// TIA Portal V15.1 export
// export: Created 2024-05-17T05:38:59.8000198Z, ExportSetting WithDefaults, DisplayName Totally Integrated Automation Portal, DisplayVersion V15.1 Update 5, DisplayName TIA Portal Openness, DisplayVersion V15.1 Update 5, DisplayName SINAMICS Startdrive Advanced, DisplayVersion V15.1, DisplayName G130, G150, S120, S150, SINAMICS MV, S210, DisplayVersion V15.1, DisplayName G110M, G120, G120C, G120D, G120P, DisplayVersion V15.1, DisplayName STEP 7 Professional, DisplayVersion V15.1 Update 5, DisplayName STEP 7 Safety, DisplayVersion V15.1, DisplayName WinCC Professional, DisplayVersion V15.1 Update 5, DisplayName SIMATIC Visualization Architect, DisplayVersion V15.1
FUNCTION "209000NCP01Config" : Void   // FC290, FBD
TITLE = 209000NCP01Config
{ S7_Optimized_Access := 'FALSE' }
AUTHOR : VCC
VERSION : 0.1
// stored: AutoNumber false, IsIECCheckEnabled false, SetENOAutomatically False, UDAEnableTagReadback false
BEGIN

REGION Network 1: **** --------------------- ETA Fuses --------------------- ****
END_REGION

REGION Network 2: **** 4.2 - Machine Status - Parameters **** AE01-JC31 // Fuse Module 1..8 (Fuse 1-16)
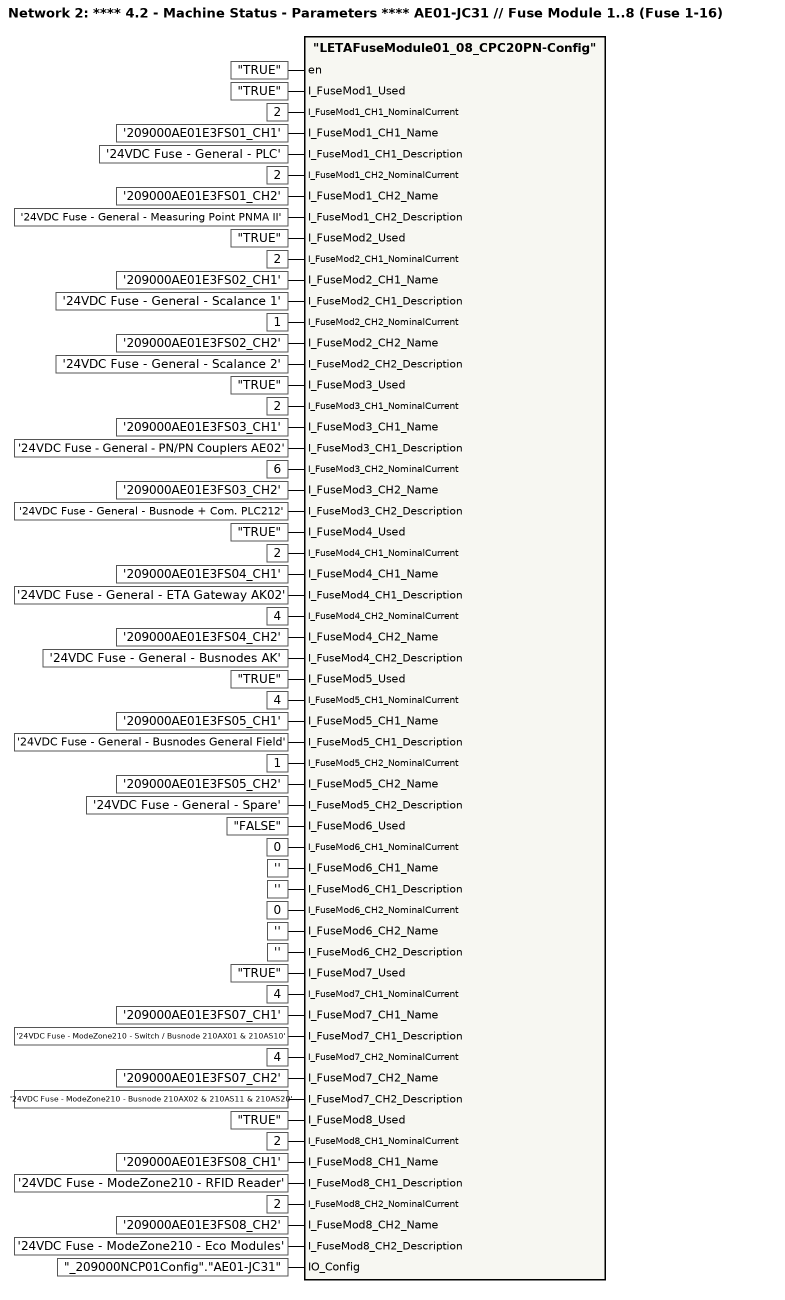
   IF "TRUE" THEN
       "LETAFuseModule01_08_CPC20PN-Config"(I_FuseMod1_Used := "TRUE",
                               I_FuseMod1_CH1_NominalCurrent := 2,
                               I_FuseMod1_CH1_Name := '209000AE01E3FS01_CH1',
                               I_FuseMod1_CH1_Description := '24VDC Fuse - General - PLC',
                               I_FuseMod1_CH2_NominalCurrent := 2,
                               I_FuseMod1_CH2_Name := '209000AE01E3FS01_CH2',
                               I_FuseMod1_CH2_Description := '24VDC Fuse - General - Measuring Point PNMA II',
                               I_FuseMod2_Used := "TRUE",
                               I_FuseMod2_CH1_NominalCurrent := 2,
                               I_FuseMod2_CH1_Name := '209000AE01E3FS02_CH1',
                               I_FuseMod2_CH1_Description := '24VDC Fuse - General - Scalance 1',
                               I_FuseMod2_CH2_NominalCurrent := 1,
                               I_FuseMod2_CH2_Name := '209000AE01E3FS02_CH2',
                               I_FuseMod2_CH2_Description := '24VDC Fuse - General - Scalance 2',
                               I_FuseMod3_Used := "TRUE",
                               I_FuseMod3_CH1_NominalCurrent := 2,
                               I_FuseMod3_CH1_Name := '209000AE01E3FS03_CH1',
                               I_FuseMod3_CH1_Description := '24VDC Fuse - General - PN/PN Couplers AE02',
                               I_FuseMod3_CH2_NominalCurrent := 6,
                               I_FuseMod3_CH2_Name := '209000AE01E3FS03_CH2',
                               I_FuseMod3_CH2_Description := '24VDC Fuse - General - Busnode + Com. PLC212',
                               I_FuseMod4_Used := "TRUE",
                               I_FuseMod4_CH1_NominalCurrent := 2,
                               I_FuseMod4_CH1_Name := '209000AE01E3FS04_CH1',
                               I_FuseMod4_CH1_Description := '24VDC Fuse - General - ETA Gateway AK02',
                               I_FuseMod4_CH2_NominalCurrent := 4,
                               I_FuseMod4_CH2_Name := '209000AE01E3FS04_CH2',
                               I_FuseMod4_CH2_Description := '24VDC Fuse - General - Busnodes AK',
                               I_FuseMod5_Used := "TRUE",
                               I_FuseMod5_CH1_NominalCurrent := 4,
                               I_FuseMod5_CH1_Name := '209000AE01E3FS05_CH1',
                               I_FuseMod5_CH1_Description := '24VDC Fuse - General - Busnodes General Field',
                               I_FuseMod5_CH2_NominalCurrent := 1,
                               I_FuseMod5_CH2_Name := '209000AE01E3FS05_CH2',
                               I_FuseMod5_CH2_Description := '24VDC Fuse - General - Spare',
                               I_FuseMod6_Used := "FALSE",
                               I_FuseMod6_CH1_NominalCurrent := 0,
                               I_FuseMod6_CH1_Name := '',
                               I_FuseMod6_CH1_Description := '',
                               I_FuseMod6_CH2_NominalCurrent := 0,
                               I_FuseMod6_CH2_Name := '',
                               I_FuseMod6_CH2_Description := '',
                               I_FuseMod7_Used := "TRUE",
                               I_FuseMod7_CH1_NominalCurrent := 4,
                               I_FuseMod7_CH1_Name := '209000AE01E3FS07_CH1',
                               I_FuseMod7_CH1_Description := '24VDC Fuse - ModeZone210 - Switch / Busnode 210AX01 & 210AS10',
                               I_FuseMod7_CH2_NominalCurrent := 4,
                               I_FuseMod7_CH2_Name := '209000AE01E3FS07_CH2',
                               I_FuseMod7_CH2_Description := '24VDC Fuse - ModeZone210 - Busnode 210AX02 & 210AS11 & 210AS20',
                               I_FuseMod8_Used := "TRUE",
                               I_FuseMod8_CH1_NominalCurrent := 2,
                               I_FuseMod8_CH1_Name := '209000AE01E3FS08_CH1',
                               I_FuseMod8_CH1_Description := '24VDC Fuse - ModeZone210 - RFID Reader',
                               I_FuseMod8_CH2_NominalCurrent := 2,
                               I_FuseMod8_CH2_Name := '209000AE01E3FS08_CH2',
                               I_FuseMod8_CH2_Description := '24VDC Fuse - ModeZone210 - Eco Modules',
                               IO_Config := "_209000NCP01Config"."AE01-JC31");
   END_IF;
END_REGION

REGION Network 3: **** 4.2 - Machine Status - Parameters **** AE01-JC31 // Fuse Module 9..16 (Fuse 17-32)
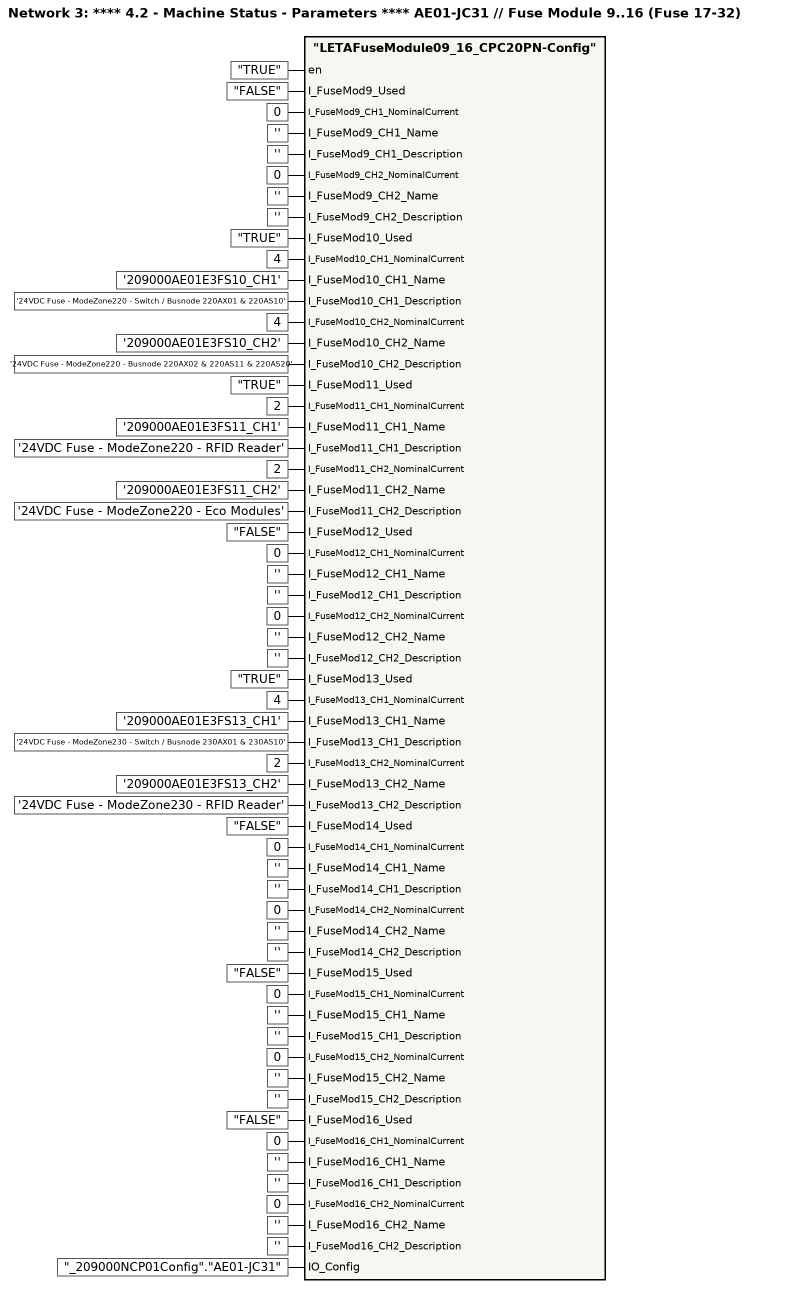
   IF "TRUE" THEN
       "LETAFuseModule09_16_CPC20PN-Config"(I_FuseMod9_Used := "FALSE",
                               I_FuseMod9_CH1_NominalCurrent := 0,
                               I_FuseMod9_CH1_Name := '',
                               I_FuseMod9_CH1_Description := '',
                               I_FuseMod9_CH2_NominalCurrent := 0,
                               I_FuseMod9_CH2_Name := '',
                               I_FuseMod9_CH2_Description := '',
                               I_FuseMod10_Used := "TRUE",
                               I_FuseMod10_CH1_NominalCurrent := 4,
                               I_FuseMod10_CH1_Name := '209000AE01E3FS10_CH1',
                               I_FuseMod10_CH1_Description := '24VDC Fuse - ModeZone220 - Switch / Busnode 220AX01 & 220AS10',
                               I_FuseMod10_CH2_NominalCurrent := 4,
                               I_FuseMod10_CH2_Name := '209000AE01E3FS10_CH2',
                               I_FuseMod10_CH2_Description := '24VDC Fuse - ModeZone220 - Busnode 220AX02 & 220AS11 & 220AS20',
                               I_FuseMod11_Used := "TRUE",
                               I_FuseMod11_CH1_NominalCurrent := 2,
                               I_FuseMod11_CH1_Name := '209000AE01E3FS11_CH1',
                               I_FuseMod11_CH1_Description := '24VDC Fuse - ModeZone220 - RFID Reader',
                               I_FuseMod11_CH2_NominalCurrent := 2,
                               I_FuseMod11_CH2_Name := '209000AE01E3FS11_CH2',
                               I_FuseMod11_CH2_Description := '24VDC Fuse - ModeZone220 - Eco Modules',
                               I_FuseMod12_Used := "FALSE",
                               I_FuseMod12_CH1_NominalCurrent := 0,
                               I_FuseMod12_CH1_Name := '',
                               I_FuseMod12_CH1_Description := '',
                               I_FuseMod12_CH2_NominalCurrent := 0,
                               I_FuseMod12_CH2_Name := '',
                               I_FuseMod12_CH2_Description := '',
                               I_FuseMod13_Used := "TRUE",
                               I_FuseMod13_CH1_NominalCurrent := 4,
                               I_FuseMod13_CH1_Name := '209000AE01E3FS13_CH1',
                               I_FuseMod13_CH1_Description := '24VDC Fuse - ModeZone230 - Switch / Busnode 230AX01 & 230AS10',
                               I_FuseMod13_CH2_NominalCurrent := 2,
                               I_FuseMod13_CH2_Name := '209000AE01E3FS13_CH2',
                               I_FuseMod13_CH2_Description := '24VDC Fuse - ModeZone230 - RFID Reader',
                               I_FuseMod14_Used := "FALSE",
                               I_FuseMod14_CH1_NominalCurrent := 0,
                               I_FuseMod14_CH1_Name := '',
                               I_FuseMod14_CH1_Description := '',
                               I_FuseMod14_CH2_NominalCurrent := 0,
                               I_FuseMod14_CH2_Name := '',
                               I_FuseMod14_CH2_Description := '',
                               I_FuseMod15_Used := "FALSE",
                               I_FuseMod15_CH1_NominalCurrent := 0,
                               I_FuseMod15_CH1_Name := '',
                               I_FuseMod15_CH1_Description := '',
                               I_FuseMod15_CH2_NominalCurrent := 0,
                               I_FuseMod15_CH2_Name := '',
                               I_FuseMod15_CH2_Description := '',
                               I_FuseMod16_Used := "FALSE",
                               I_FuseMod16_CH1_NominalCurrent := 0,
                               I_FuseMod16_CH1_Name := '',
                               I_FuseMod16_CH1_Description := '',
                               I_FuseMod16_CH2_NominalCurrent := 0,
                               I_FuseMod16_CH2_Name := '',
                               I_FuseMod16_CH2_Description := '',
                               IO_Config := "_209000NCP01Config"."AE01-JC31");
   END_IF;
END_REGION

REGION Network 4: **** 4.2 - Machine Status - Parameters **** AK02-JC32 // Fuse Module 1..8 (Fuse 1-16)
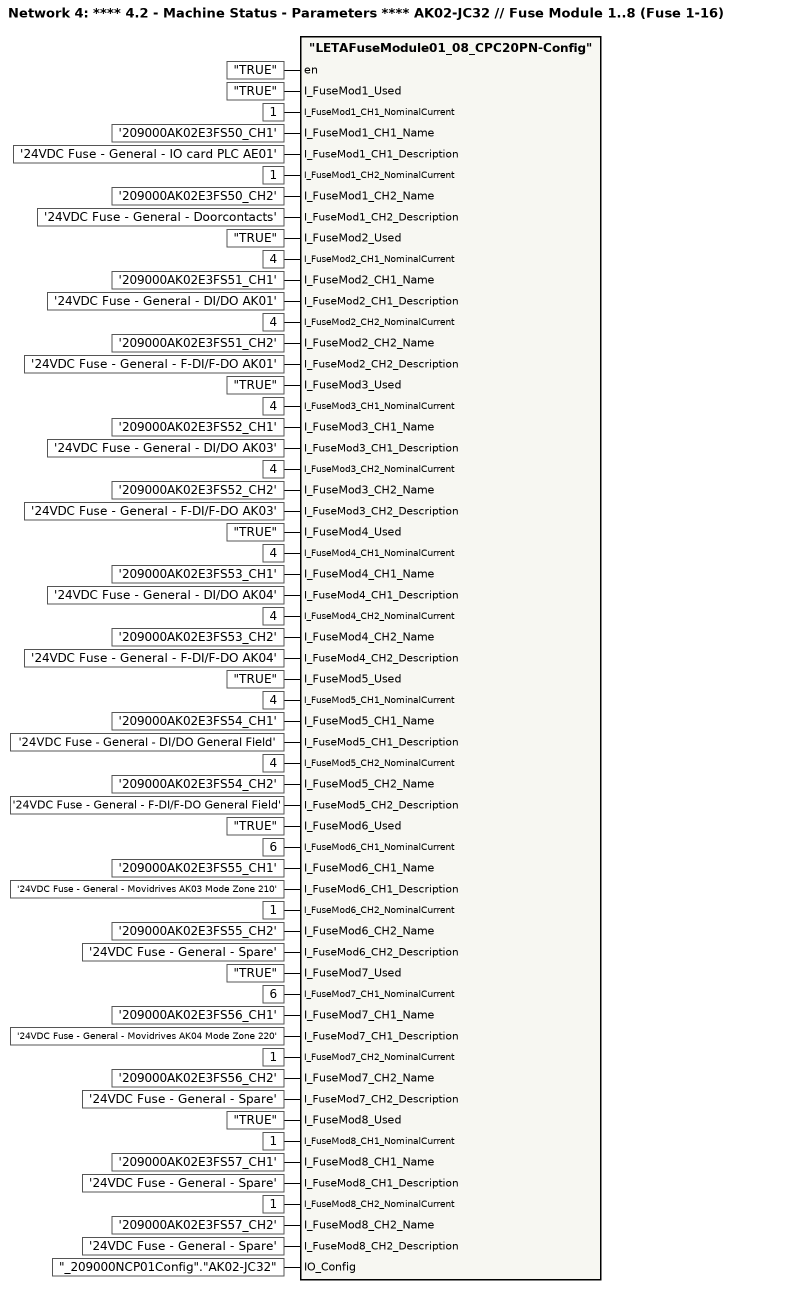
   IF "TRUE" THEN
       "LETAFuseModule01_08_CPC20PN-Config"(I_FuseMod1_Used := "TRUE",
                               I_FuseMod1_CH1_NominalCurrent := 1,
                               I_FuseMod1_CH1_Name := '209000AK02E3FS50_CH1',
                               I_FuseMod1_CH1_Description := '24VDC Fuse - General - IO card PLC AE01',
                               I_FuseMod1_CH2_NominalCurrent := 1,
                               I_FuseMod1_CH2_Name := '209000AK02E3FS50_CH2',
                               I_FuseMod1_CH2_Description := '24VDC Fuse - General - Doorcontacts',
                               I_FuseMod2_Used := "TRUE",
                               I_FuseMod2_CH1_NominalCurrent := 4,
                               I_FuseMod2_CH1_Name := '209000AK02E3FS51_CH1',
                               I_FuseMod2_CH1_Description := '24VDC Fuse - General - DI/DO AK01',
                               I_FuseMod2_CH2_NominalCurrent := 4,
                               I_FuseMod2_CH2_Name := '209000AK02E3FS51_CH2',
                               I_FuseMod2_CH2_Description := '24VDC Fuse - General - F-DI/F-DO AK01',
                               I_FuseMod3_Used := "TRUE",
                               I_FuseMod3_CH1_NominalCurrent := 4,
                               I_FuseMod3_CH1_Name := '209000AK02E3FS52_CH1',
                               I_FuseMod3_CH1_Description := '24VDC Fuse - General - DI/DO AK03',
                               I_FuseMod3_CH2_NominalCurrent := 4,
                               I_FuseMod3_CH2_Name := '209000AK02E3FS52_CH2',
                               I_FuseMod3_CH2_Description := '24VDC Fuse - General - F-DI/F-DO AK03',
                               I_FuseMod4_Used := "TRUE",
                               I_FuseMod4_CH1_NominalCurrent := 4,
                               I_FuseMod4_CH1_Name := '209000AK02E3FS53_CH1',
                               I_FuseMod4_CH1_Description := '24VDC Fuse - General - DI/DO AK04',
                               I_FuseMod4_CH2_NominalCurrent := 4,
                               I_FuseMod4_CH2_Name := '209000AK02E3FS53_CH2',
                               I_FuseMod4_CH2_Description := '24VDC Fuse - General - F-DI/F-DO AK04',
                               I_FuseMod5_Used := "TRUE",
                               I_FuseMod5_CH1_NominalCurrent := 4,
                               I_FuseMod5_CH1_Name := '209000AK02E3FS54_CH1',
                               I_FuseMod5_CH1_Description := '24VDC Fuse - General - DI/DO General Field',
                               I_FuseMod5_CH2_NominalCurrent := 4,
                               I_FuseMod5_CH2_Name := '209000AK02E3FS54_CH2',
                               I_FuseMod5_CH2_Description := '24VDC Fuse - General - F-DI/F-DO General Field',
                               I_FuseMod6_Used := "TRUE",
                               I_FuseMod6_CH1_NominalCurrent := 6,
                               I_FuseMod6_CH1_Name := '209000AK02E3FS55_CH1',
                               I_FuseMod6_CH1_Description := '24VDC Fuse - General - Movidrives AK03 Mode Zone 210',
                               I_FuseMod6_CH2_NominalCurrent := 1,
                               I_FuseMod6_CH2_Name := '209000AK02E3FS55_CH2',
                               I_FuseMod6_CH2_Description := '24VDC Fuse - General - Spare',
                               I_FuseMod7_Used := "TRUE",
                               I_FuseMod7_CH1_NominalCurrent := 6,
                               I_FuseMod7_CH1_Name := '209000AK02E3FS56_CH1',
                               I_FuseMod7_CH1_Description := '24VDC Fuse - General - Movidrives AK04 Mode Zone 220',
                               I_FuseMod7_CH2_NominalCurrent := 1,
                               I_FuseMod7_CH2_Name := '209000AK02E3FS56_CH2',
                               I_FuseMod7_CH2_Description := '24VDC Fuse - General - Spare',
                               I_FuseMod8_Used := "TRUE",
                               I_FuseMod8_CH1_NominalCurrent := 1,
                               I_FuseMod8_CH1_Name := '209000AK02E3FS57_CH1',
                               I_FuseMod8_CH1_Description := '24VDC Fuse - General - Spare',
                               I_FuseMod8_CH2_NominalCurrent := 1,
                               I_FuseMod8_CH2_Name := '209000AK02E3FS57_CH2',
                               I_FuseMod8_CH2_Description := '24VDC Fuse - General - Spare',
                               IO_Config := "_209000NCP01Config"."AK02-JC32");
   END_IF;
END_REGION

REGION Network 5: **** 4.2 - Machine Status - Parameters **** AK02-JC32 // Fuse Module 9..16 (Fuse 17-32)
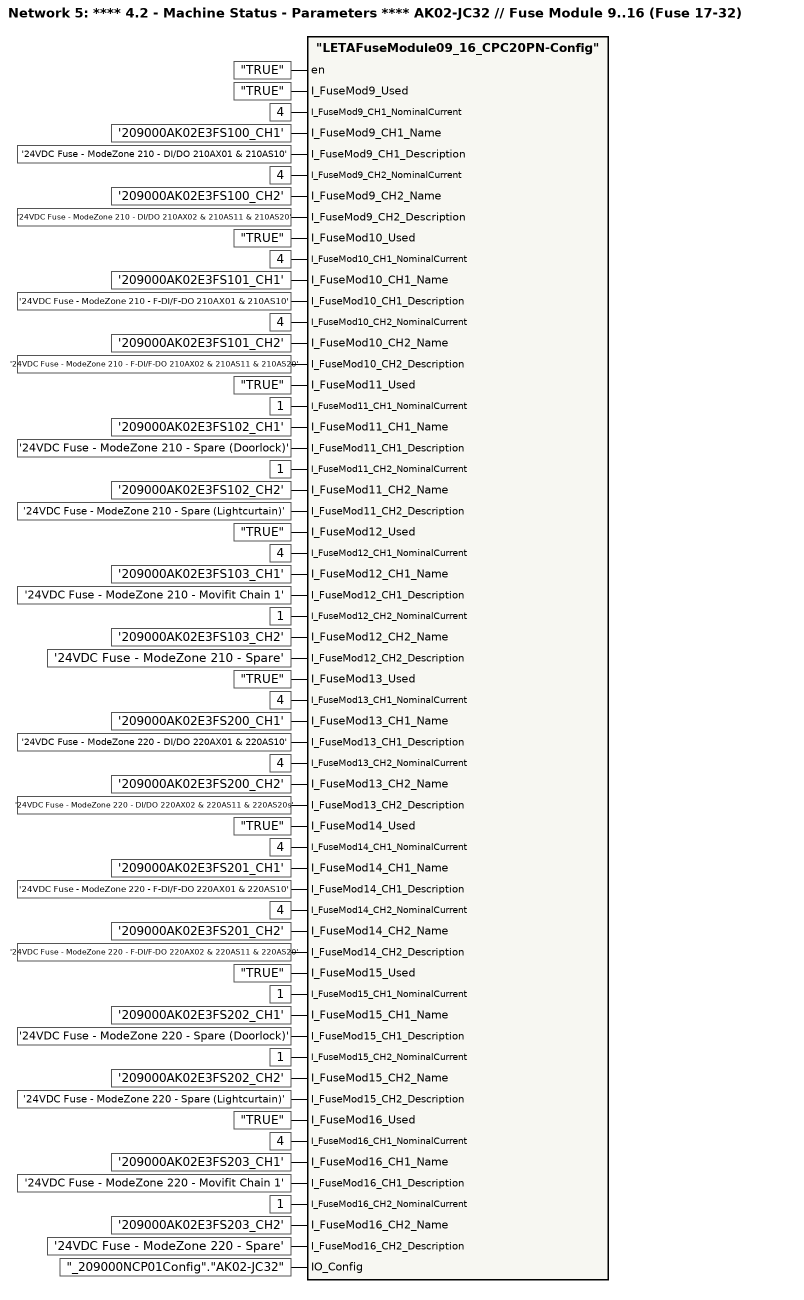
   IF "TRUE" THEN
       "LETAFuseModule09_16_CPC20PN-Config"(I_FuseMod9_Used := "TRUE",
                               I_FuseMod9_CH1_NominalCurrent := 4,
                               I_FuseMod9_CH1_Name := '209000AK02E3FS100_CH1',
                               I_FuseMod9_CH1_Description := '24VDC Fuse - ModeZone 210 - DI/DO 210AX01 & 210AS10',
                               I_FuseMod9_CH2_NominalCurrent := 4,
                               I_FuseMod9_CH2_Name := '209000AK02E3FS100_CH2',
                               I_FuseMod9_CH2_Description := '24VDC Fuse - ModeZone 210 - DI/DO 210AX02 & 210AS11 & 210AS20',
                               I_FuseMod10_Used := "TRUE",
                               I_FuseMod10_CH1_NominalCurrent := 4,
                               I_FuseMod10_CH1_Name := '209000AK02E3FS101_CH1',
                               I_FuseMod10_CH1_Description := '24VDC Fuse - ModeZone 210 - F-DI/F-DO 210AX01 & 210AS10',
                               I_FuseMod10_CH2_NominalCurrent := 4,
                               I_FuseMod10_CH2_Name := '209000AK02E3FS101_CH2',
                               I_FuseMod10_CH2_Description := '24VDC Fuse - ModeZone 210 - F-DI/F-DO 210AX02 & 210AS11 & 210AS20',
                               I_FuseMod11_Used := "TRUE",
                               I_FuseMod11_CH1_NominalCurrent := 1,
                               I_FuseMod11_CH1_Name := '209000AK02E3FS102_CH1',
                               I_FuseMod11_CH1_Description := '24VDC Fuse - ModeZone 210 - Spare (Doorlock)',
                               I_FuseMod11_CH2_NominalCurrent := 1,
                               I_FuseMod11_CH2_Name := '209000AK02E3FS102_CH2',
                               I_FuseMod11_CH2_Description := '24VDC Fuse - ModeZone 210 - Spare (Lightcurtain)',
                               I_FuseMod12_Used := "TRUE",
                               I_FuseMod12_CH1_NominalCurrent := 4,
                               I_FuseMod12_CH1_Name := '209000AK02E3FS103_CH1',
                               I_FuseMod12_CH1_Description := '24VDC Fuse - ModeZone 210 - Movifit Chain 1',
                               I_FuseMod12_CH2_NominalCurrent := 1,
                               I_FuseMod12_CH2_Name := '209000AK02E3FS103_CH2',
                               I_FuseMod12_CH2_Description := '24VDC Fuse - ModeZone 210 - Spare',
                               I_FuseMod13_Used := "TRUE",
                               I_FuseMod13_CH1_NominalCurrent := 4,
                               I_FuseMod13_CH1_Name := '209000AK02E3FS200_CH1',
                               I_FuseMod13_CH1_Description := '24VDC Fuse - ModeZone 220 - DI/DO 220AX01 & 220AS10',
                               I_FuseMod13_CH2_NominalCurrent := 4,
                               I_FuseMod13_CH2_Name := '209000AK02E3FS200_CH2',
                               I_FuseMod13_CH2_Description := '24VDC Fuse - ModeZone 220 - DI/DO 220AX02 & 220AS11 & 220AS20s',
                               I_FuseMod14_Used := "TRUE",
                               I_FuseMod14_CH1_NominalCurrent := 4,
                               I_FuseMod14_CH1_Name := '209000AK02E3FS201_CH1',
                               I_FuseMod14_CH1_Description := '24VDC Fuse - ModeZone 220 - F-DI/F-DO 220AX01 & 220AS10',
                               I_FuseMod14_CH2_NominalCurrent := 4,
                               I_FuseMod14_CH2_Name := '209000AK02E3FS201_CH2',
                               I_FuseMod14_CH2_Description := '24VDC Fuse - ModeZone 220 - F-DI/F-DO 220AX02 & 220AS11 & 220AS20',
                               I_FuseMod15_Used := "TRUE",
                               I_FuseMod15_CH1_NominalCurrent := 1,
                               I_FuseMod15_CH1_Name := '209000AK02E3FS202_CH1',
                               I_FuseMod15_CH1_Description := '24VDC Fuse - ModeZone 220 - Spare (Doorlock)',
                               I_FuseMod15_CH2_NominalCurrent := 1,
                               I_FuseMod15_CH2_Name := '209000AK02E3FS202_CH2',
                               I_FuseMod15_CH2_Description := '24VDC Fuse - ModeZone 220 - Spare (Lightcurtain)',
                               I_FuseMod16_Used := "TRUE",
                               I_FuseMod16_CH1_NominalCurrent := 4,
                               I_FuseMod16_CH1_Name := '209000AK02E3FS203_CH1',
                               I_FuseMod16_CH1_Description := '24VDC Fuse - ModeZone 220 - Movifit Chain 1',
                               I_FuseMod16_CH2_NominalCurrent := 1,
                               I_FuseMod16_CH2_Name := '209000AK02E3FS203_CH2',
                               I_FuseMod16_CH2_Description := '24VDC Fuse - ModeZone 220 - Spare',
                               IO_Config := "_209000NCP01Config"."AK02-JC32");
   END_IF;
END_REGION

REGION Network 6: **** 4.2 - Machine Status - Parameters **** AK02-JC32 // Fuse Module 17..24 (Fuse 33-48)
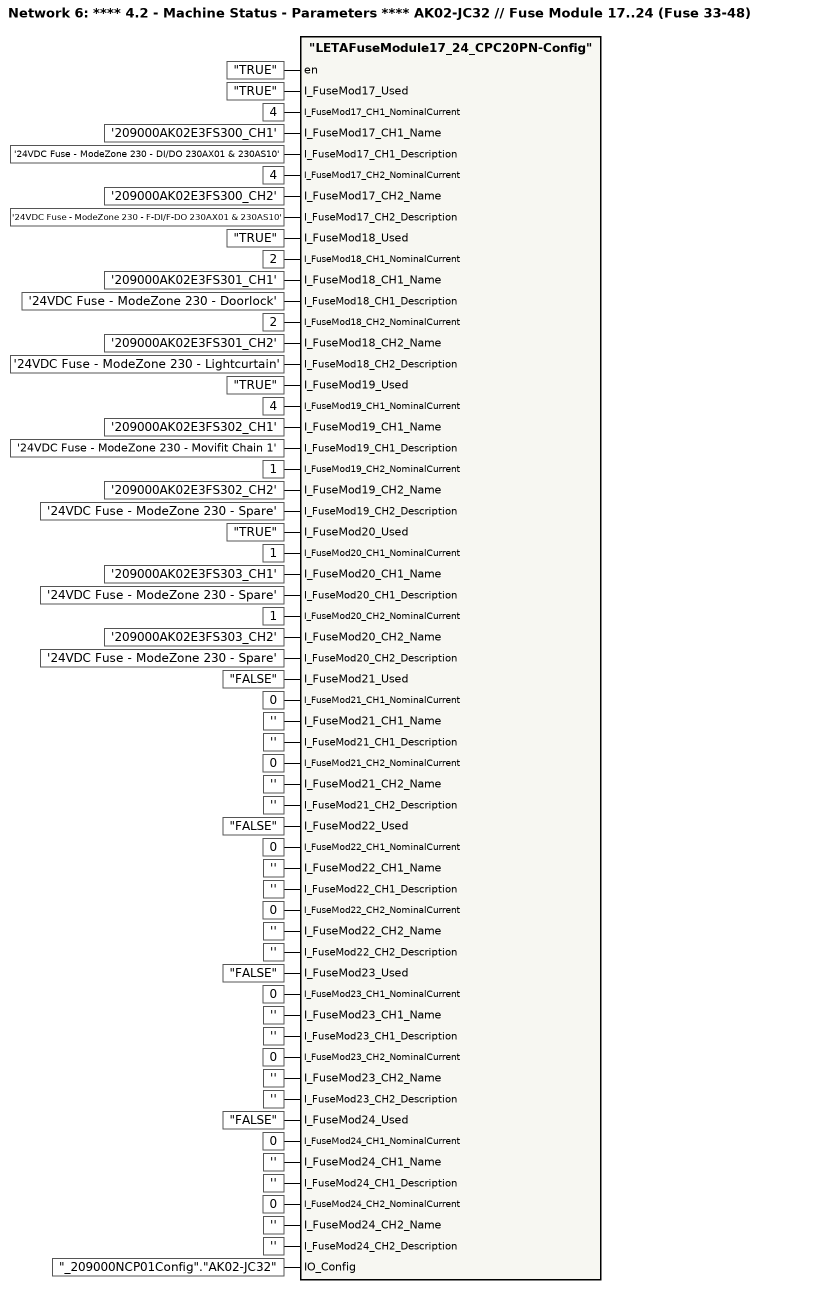
   IF "TRUE" THEN
       "LETAFuseModule17_24_CPC20PN-Config"(I_FuseMod17_Used := "TRUE",
                               I_FuseMod17_CH1_NominalCurrent := 4,
                               I_FuseMod17_CH1_Name := '209000AK02E3FS300_CH1',
                               I_FuseMod17_CH1_Description := '24VDC Fuse - ModeZone 230 - DI/DO 230AX01 & 230AS10',
                               I_FuseMod17_CH2_NominalCurrent := 4,
                               I_FuseMod17_CH2_Name := '209000AK02E3FS300_CH2',
                               I_FuseMod17_CH2_Description := '24VDC Fuse - ModeZone 230 - F-DI/F-DO 230AX01 & 230AS10',
                               I_FuseMod18_Used := "TRUE",
                               I_FuseMod18_CH1_NominalCurrent := 2,
                               I_FuseMod18_CH1_Name := '209000AK02E3FS301_CH1',
                               I_FuseMod18_CH1_Description := '24VDC Fuse - ModeZone 230 - Doorlock',
                               I_FuseMod18_CH2_NominalCurrent := 2,
                               I_FuseMod18_CH2_Name := '209000AK02E3FS301_CH2',
                               I_FuseMod18_CH2_Description := '24VDC Fuse - ModeZone 230 - Lightcurtain',
                               I_FuseMod19_Used := "TRUE",
                               I_FuseMod19_CH1_NominalCurrent := 4,
                               I_FuseMod19_CH1_Name := '209000AK02E3FS302_CH1',
                               I_FuseMod19_CH1_Description := '24VDC Fuse - ModeZone 230 - Movifit Chain 1',
                               I_FuseMod19_CH2_NominalCurrent := 1,
                               I_FuseMod19_CH2_Name := '209000AK02E3FS302_CH2',
                               I_FuseMod19_CH2_Description := '24VDC Fuse - ModeZone 230 - Spare',
                               I_FuseMod20_Used := "TRUE",
                               I_FuseMod20_CH1_NominalCurrent := 1,
                               I_FuseMod20_CH1_Name := '209000AK02E3FS303_CH1',
                               I_FuseMod20_CH1_Description := '24VDC Fuse - ModeZone 230 - Spare',
                               I_FuseMod20_CH2_NominalCurrent := 1,
                               I_FuseMod20_CH2_Name := '209000AK02E3FS303_CH2',
                               I_FuseMod20_CH2_Description := '24VDC Fuse - ModeZone 230 - Spare',
                               I_FuseMod21_Used := "FALSE",
                               I_FuseMod21_CH1_NominalCurrent := 0,
                               I_FuseMod21_CH1_Name := '',
                               I_FuseMod21_CH1_Description := '',
                               I_FuseMod21_CH2_NominalCurrent := 0,
                               I_FuseMod21_CH2_Name := '',
                               I_FuseMod21_CH2_Description := '',
                               I_FuseMod22_Used := "FALSE",
                               I_FuseMod22_CH1_NominalCurrent := 0,
                               I_FuseMod22_CH1_Name := '',
                               I_FuseMod22_CH1_Description := '',
                               I_FuseMod22_CH2_NominalCurrent := 0,
                               I_FuseMod22_CH2_Name := '',
                               I_FuseMod22_CH2_Description := '',
                               I_FuseMod23_Used := "FALSE",
                               I_FuseMod23_CH1_NominalCurrent := 0,
                               I_FuseMod23_CH1_Name := '',
                               I_FuseMod23_CH1_Description := '',
                               I_FuseMod23_CH2_NominalCurrent := 0,
                               I_FuseMod23_CH2_Name := '',
                               I_FuseMod23_CH2_Description := '',
                               I_FuseMod24_Used := "FALSE",
                               I_FuseMod24_CH1_NominalCurrent := 0,
                               I_FuseMod24_CH1_Name := '',
                               I_FuseMod24_CH1_Description := '',
                               I_FuseMod24_CH2_NominalCurrent := 0,
                               I_FuseMod24_CH2_Name := '',
                               I_FuseMod24_CH2_Description := '',
                               IO_Config := "_209000NCP01Config"."AK02-JC32");
   END_IF;
END_REGION

REGION Network 7: **** 4.2 - Machine Status - Parameters **** AK02-JC32 // Fuse Module 25..32 (Fuse 49-64)
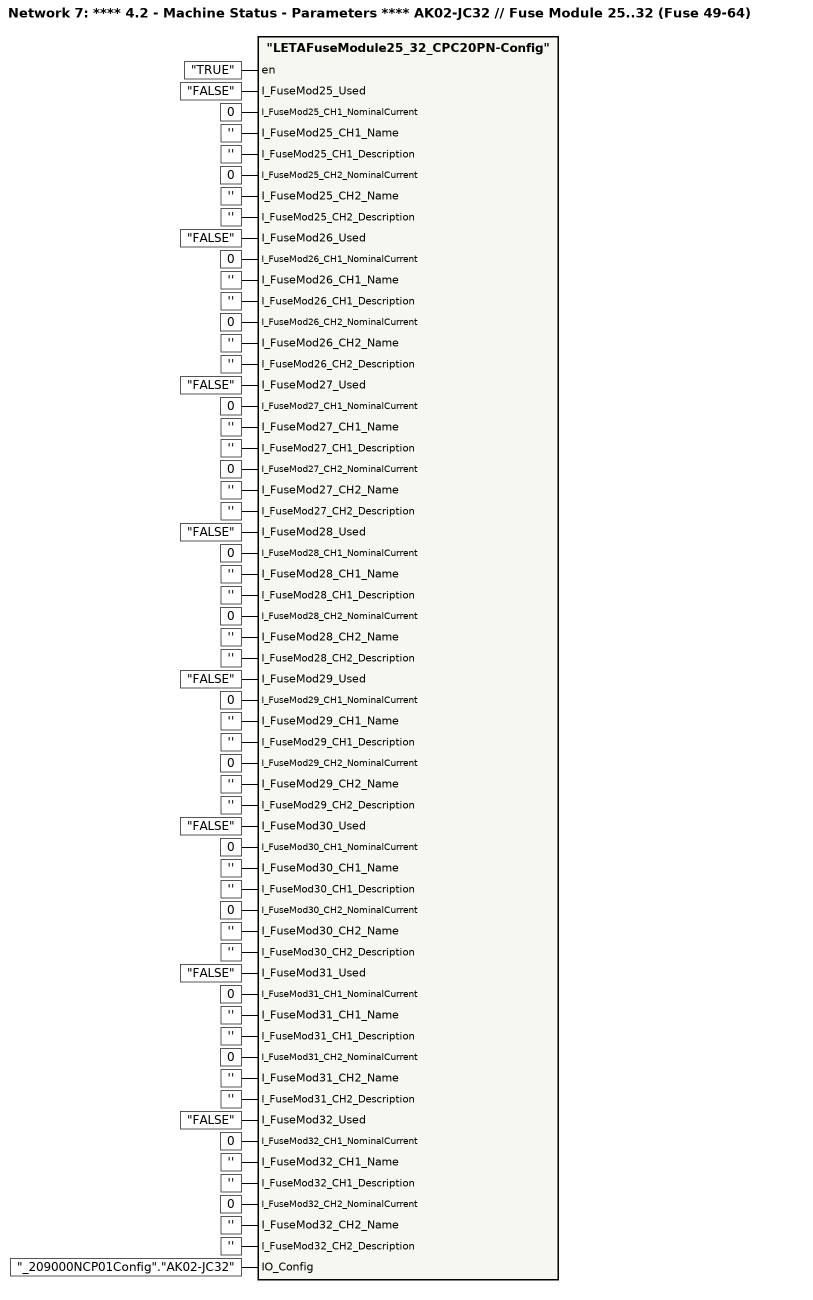
   IF "TRUE" THEN
       "LETAFuseModule25_32_CPC20PN-Config"(I_FuseMod25_Used := "FALSE",
                               I_FuseMod25_CH1_NominalCurrent := 0,
                               I_FuseMod25_CH1_Name := '',
                               I_FuseMod25_CH1_Description := '',
                               I_FuseMod25_CH2_NominalCurrent := 0,
                               I_FuseMod25_CH2_Name := '',
                               I_FuseMod25_CH2_Description := '',
                               I_FuseMod26_Used := "FALSE",
                               I_FuseMod26_CH1_NominalCurrent := 0,
                               I_FuseMod26_CH1_Name := '',
                               I_FuseMod26_CH1_Description := '',
                               I_FuseMod26_CH2_NominalCurrent := 0,
                               I_FuseMod26_CH2_Name := '',
                               I_FuseMod26_CH2_Description := '',
                               I_FuseMod27_Used := "FALSE",
                               I_FuseMod27_CH1_NominalCurrent := 0,
                               I_FuseMod27_CH1_Name := '',
                               I_FuseMod27_CH1_Description := '',
                               I_FuseMod27_CH2_NominalCurrent := 0,
                               I_FuseMod27_CH2_Name := '',
                               I_FuseMod27_CH2_Description := '',
                               I_FuseMod28_Used := "FALSE",
                               I_FuseMod28_CH1_NominalCurrent := 0,
                               I_FuseMod28_CH1_Name := '',
                               I_FuseMod28_CH1_Description := '',
                               I_FuseMod28_CH2_NominalCurrent := 0,
                               I_FuseMod28_CH2_Name := '',
                               I_FuseMod28_CH2_Description := '',
                               I_FuseMod29_Used := "FALSE",
                               I_FuseMod29_CH1_NominalCurrent := 0,
                               I_FuseMod29_CH1_Name := '',
                               I_FuseMod29_CH1_Description := '',
                               I_FuseMod29_CH2_NominalCurrent := 0,
                               I_FuseMod29_CH2_Name := '',
                               I_FuseMod29_CH2_Description := '',
                               I_FuseMod30_Used := "FALSE",
                               I_FuseMod30_CH1_NominalCurrent := 0,
                               I_FuseMod30_CH1_Name := '',
                               I_FuseMod30_CH1_Description := '',
                               I_FuseMod30_CH2_NominalCurrent := 0,
                               I_FuseMod30_CH2_Name := '',
                               I_FuseMod30_CH2_Description := '',
                               I_FuseMod31_Used := "FALSE",
                               I_FuseMod31_CH1_NominalCurrent := 0,
                               I_FuseMod31_CH1_Name := '',
                               I_FuseMod31_CH1_Description := '',
                               I_FuseMod31_CH2_NominalCurrent := 0,
                               I_FuseMod31_CH2_Name := '',
                               I_FuseMod31_CH2_Description := '',
                               I_FuseMod32_Used := "FALSE",
                               I_FuseMod32_CH1_NominalCurrent := 0,
                               I_FuseMod32_CH1_Name := '',
                               I_FuseMod32_CH1_Description := '',
                               I_FuseMod32_CH2_NominalCurrent := 0,
                               I_FuseMod32_CH2_Name := '',
                               I_FuseMod32_CH2_Description := '',
                               IO_Config := "_209000NCP01Config"."AK02-JC32");
   END_IF;
END_REGION
END_FUNCTION
